{attribute 'pack_mode' := '1'}
TYPE TRunDataPlate :
STRUCT
	ePartStatus	: TPlatePartStatus;
END_STRUCT
END_TYPE

(* stored: Version 1.1.0.1, ProductVersion 3.1.4022.12
   DUT TRunDataPlate: Id {ca9e88ea-d843-43e4-85ff-cedc0f3e6739} *)
